VISUALIZATION Visualization  // 2x2
END_VISUALIZATION

(* stored: Version 1.1.0.1, ProductVersion 3.1.4024.15
   Visu Visualization: Id {531e480f-00cc-47bb-9fa3-160da29ffcad} *)
